// Mitsubishi GX Works2 project: 2023-06-14 #1 생산자동화기능사 8번   PLC: Q03UDV
// 생산자동화기능사

// global labels: Global1
VAR_GLOBAL
  PB1 AT X0 : BOOL;
  PB2 AT X1 : BOOL;
  정지 AT X2 : BOOL;
  공급후진 AT X3 : BOOL;
  공급전진 AT X4 : BOOL;
  가공후진 AT X5 : BOOL;
  가공전진 AT X6 : BOOL;
  송출후진 AT X7 : BOOL;
  송출전진 AT X8 : BOOL;
  배출후진 AT X9 : BOOL;
  배출전진 AT X0A : BOOL;
  매거진 AT X0B : BOOL;
  금속센서 AT X0F : BOOL;
  PB3 AT X10 : BOOL;
  적색 AT Y20 : BOOL;
  황색 AT Y21 : BOOL;
  녹색 AT Y22 : BOOL;
  공급1 AT Y23 : BOOL;
  공급2 AT Y24 : BOOL;
  가공 AT Y25 : BOOL;
  드릴 AT Y26 : BOOL;
  송출 AT Y27 : BOOL;
  배출 AT Y28 : BOOL;
  컨베이어 AT Y29 : BOOL;
END_VAR

PROGRAM 테스트동작
VAR
  PHASE : INT;
END_VAR
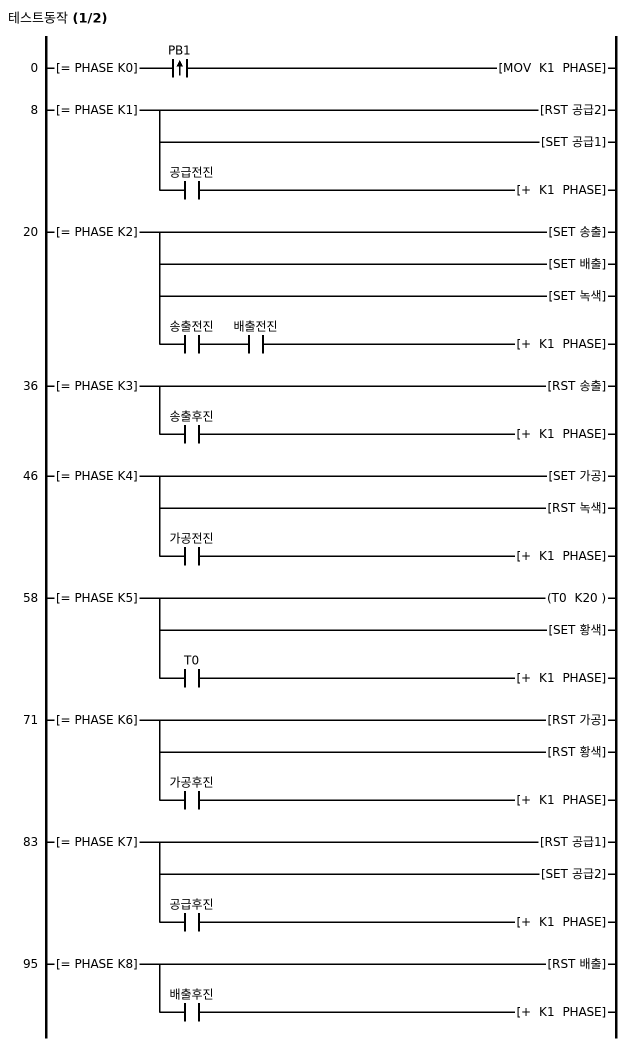
0     LD=     PHASE K0
      ANDP    PB1
      MOV     K1 PHASE
8     LD=     PHASE K1
      RST     공급2
      SET     공급1
      AND     공급전진
      +       K1 PHASE
20    LD=     PHASE K2
      SET     송출
      SET     배출
      SET     녹색
      AND     송출전진
      AND     배출전진
      +       K1 PHASE
36    LD=     PHASE K3
      RST     송출
      AND     송출후진
      +       K1 PHASE
46    LD=     PHASE K4
      SET     가공
      RST     녹색
      AND     가공전진
      +       K1 PHASE
58    LD=     PHASE K5
      OUT     T0 K20
      SET     황색
      AND     T0
      +       K1 PHASE
71    LD=     PHASE K6
      RST     가공
      RST     황색
      AND     가공후진
      +       K1 PHASE
83    LD=     PHASE K7
      RST     공급1
      SET     공급2
      AND     공급후진
      +       K1 PHASE
95    LD=     PHASE K8
      RST     배출
      AND     배출후진
      +       K1 PHASE
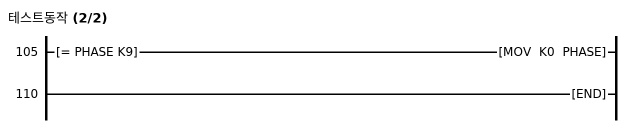
105   LD=     PHASE K9
      MOV     K0 PHASE
110   END
END_PROGRAM

PROGRAM 생산자동화기능사
VAR
  PHASE : INT;
  MODE : INT;
END_VAR
VAR CONSTANT
  단속 : INT;
  연속 : INT := 1;
END_VAR
VAR
  EMG : BOOL;
  BLINK : ARRAY [0..3] OF BOOL;
  PHASE1 : INT;
END_VAR
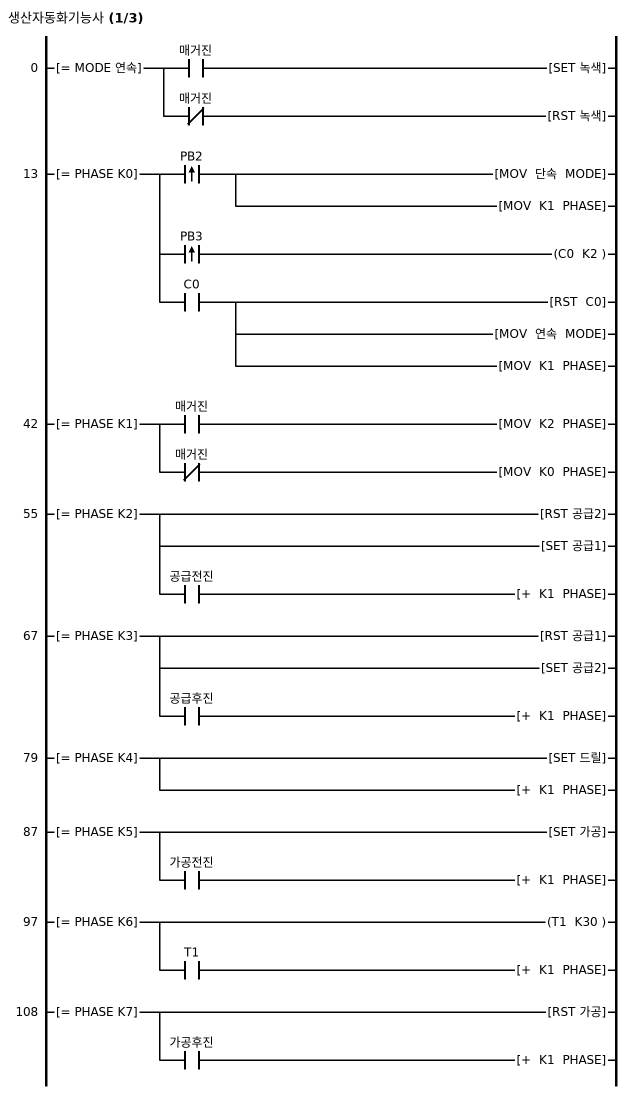
0     LD=     MODE 연속
      MPS
      AND     매거진
      SET     녹색
      MPP
      ANI     매거진
      RST     녹색
13    LD=     PHASE K0
      MPS
      ANDP    PB2
      MOV     단속 MODE
      MOV     K1 PHASE
      MRD
      ANDP    PB3
      OUT     C0 K2
      MPP
      AND     C0
      RST     C0
      MOV     연속 MODE
      MOV     K1 PHASE
42    LD=     PHASE K1
      MPS
      AND     매거진
      MOV     K2 PHASE
      MPP
      ANI     매거진
      MOV     K0 PHASE
55    LD=     PHASE K2
      RST     공급2
      SET     공급1
      AND     공급전진
      +       K1 PHASE
67    LD=     PHASE K3
      RST     공급1
      SET     공급2
      AND     공급후진
      +       K1 PHASE
79    LD=     PHASE K4
      SET     드릴
      +       K1 PHASE
87    LD=     PHASE K5
      SET     가공
      AND     가공전진
      +       K1 PHASE
97    LD=     PHASE K6
      OUT     T1 K30
      AND     T1
      +       K1 PHASE
108   LD=     PHASE K7
      RST     가공
      AND     가공후진
      +       K1 PHASE
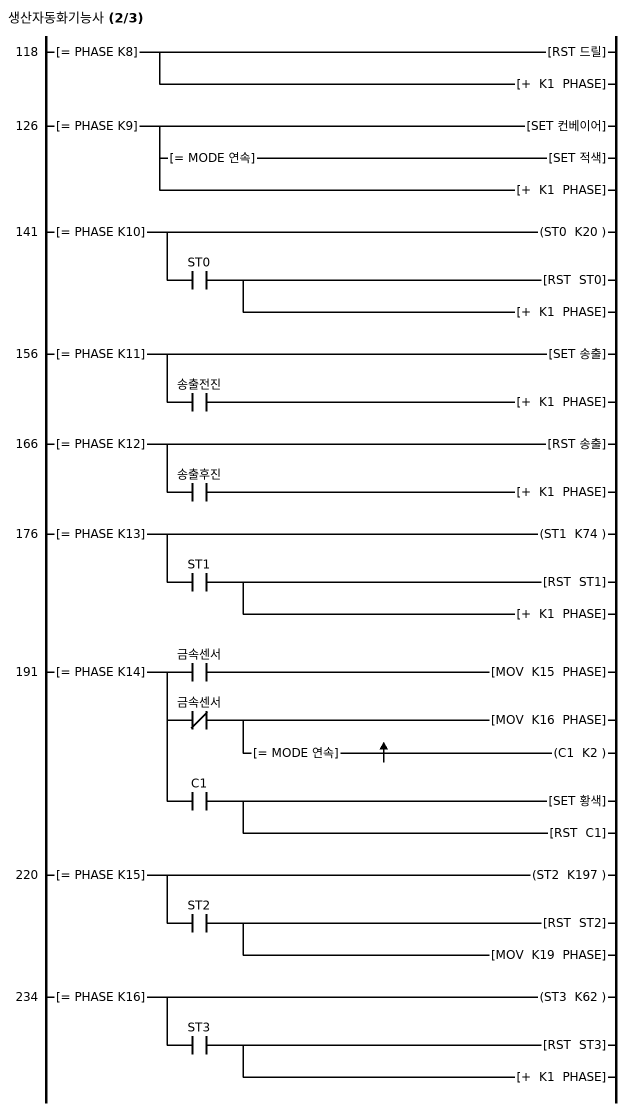
118   LD=     PHASE K8
      RST     드릴
      +       K1 PHASE
126   LD=     PHASE K9
      SET     컨베이어
      MPS
      AND=    MODE 연속
      SET     적색
      MPP
      +       K1 PHASE
141   LD=     PHASE K10
      OUT     ST0 K20
      AND     ST0
      RST     ST0
      +       K1 PHASE
156   LD=     PHASE K11
      SET     송출
      AND     송출전진
      +       K1 PHASE
166   LD=     PHASE K12
      RST     송출
      AND     송출후진
      +       K1 PHASE
176   LD=     PHASE K13
      OUT     ST1 K74
      AND     ST1
      RST     ST1
      +       K1 PHASE
191   LD=     PHASE K14
      MPS
      AND     금속센서
      MOV     K15 PHASE
      MRD
      ANI     금속센서
      MOV     K16 PHASE
      AND=    MODE 연속
      MEP
      OUT     C1 K2
      MPP
      AND     C1
      SET     황색
      RST     C1
220   LD=     PHASE K15
      OUT     ST2 K197
      AND     ST2
      RST     ST2
      MOV     K19 PHASE
234   LD=     PHASE K16
      OUT     ST3 K62
      AND     ST3
      RST     ST3
      +       K1 PHASE
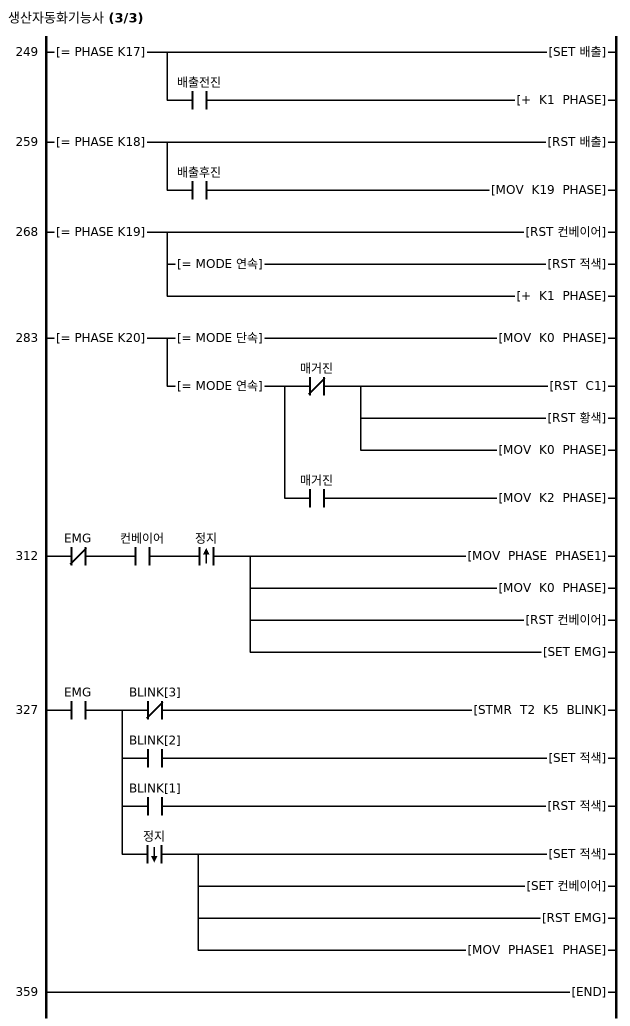
249   LD=     PHASE K17
      SET     배출
      AND     배출전진
      +       K1 PHASE
259   LD=     PHASE K18
      RST     배출
      AND     배출후진
      MOV     K19 PHASE
268   LD=     PHASE K19
      RST     컨베이어
      MPS
      AND=    MODE 연속
      RST     적색
      MPP
      +       K1 PHASE
283   LD=     PHASE K20
      MPS
      AND=    MODE 단속
      MOV     K0 PHASE
      MPP
      AND=    MODE 연속
      MPS
      ANI     매거진
      RST     C1
      RST     황색
      MOV     K0 PHASE
      MPP
      AND     매거진
      MOV     K2 PHASE
312   LDI     EMG
      AND     컨베이어
      ANDP    정지
      MOV     PHASE PHASE1
      MOV     K0 PHASE
      RST     컨베이어
      SET     EMG
327   LD      EMG
      MPS
      ANI     BLINK[3]
      STMR    T2 K5 BLINK
      MRD
      AND     BLINK[2]
      SET     적색
      MRD
      AND     BLINK[1]
      RST     적색
      MPP
      ANDF    정지
      SET     적색
      SET     컨베이어
      RST     EMG
      MOV     PHASE1 PHASE
359   END
END_PROGRAM
